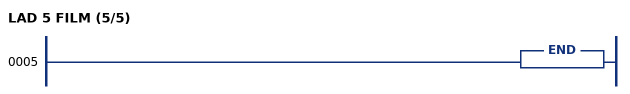
% Rung: 5 %
SOR END EOR

LADDER 6 "PROFILES"
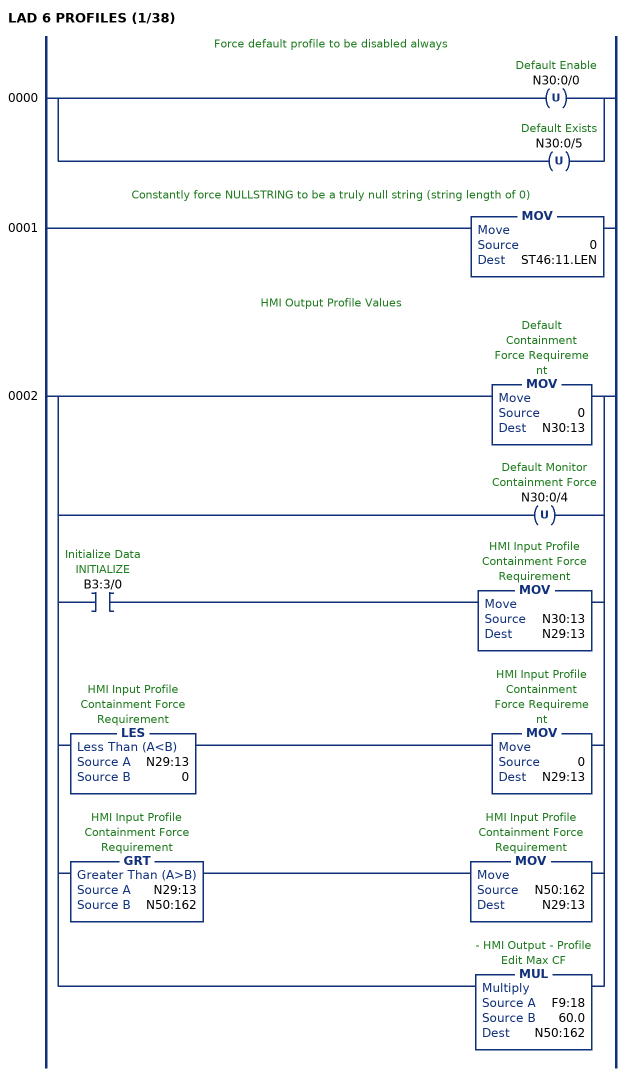
% Rung: 0 %
% Force default profile to be disabled always %
SOR BST OTU N30:0/0 NXB OTU N30:0/5 BND EOR
%   N30:0/0  "Default Enable" %
%   N30:0/5  "Default Exists" %
% Rung: 1 %
% Constantly force NULLSTRING to be a truly null string (string length of 0) %
SOR MOV 0 ST46:11.LEN EOR
% Rung: 2 %
% HMI Output Profile Values %
SOR BST MOV 0 N30:13 NXB OTU N30:0/4 NXB XIC B3:3/0 MOV N30:13 N29:13 NXB LES N29:13 0 MOV 0 N29:13 NXB GRT N29:13 N50:162 MOV N50:162 N29:13 NXB MUL F9:18 60.0 N50:162 BND EOR
%   N30:13  "Default Containment Force Requirement" %
%   N30:0/4  "Default Monitor Containment Force" %
%   B3:3/0  INITIALIZE  "Initialize Data" %
%   N29:13  "HMI Input Profile Containment Force Requirement" %
%   N50:162  "- HMI Output - Profile Edit Max CF" %
%   F9:18  INCREMENTALAT15  "Incremental CF At WF15 For A Given Film Thickness" %

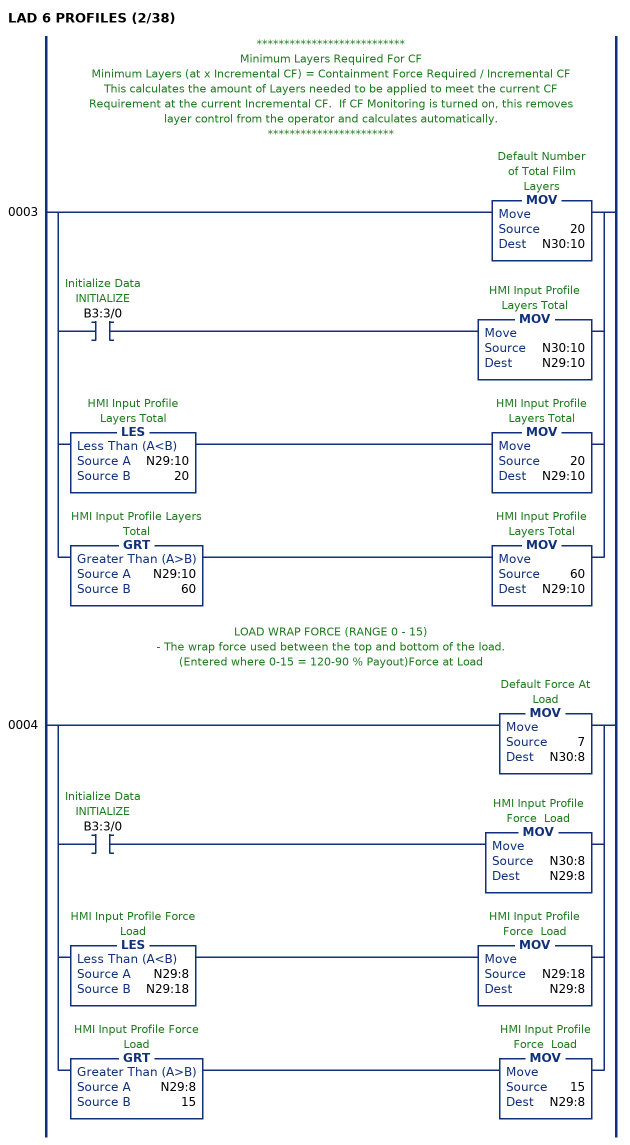
% Rung: 3 %
% ***************************
% 
% Minimum Layers Required For CF
% 
% Minimum Layers (at x Incremental CF) = Containment Force Required / Incremental CF
% 
% This calculates the amount of Layers needed to be applied to meet the current CF Requirement at the current Incremental CF.  If CF Monitoring is turned on, this removes layer control from the operator and calculates automatically.
% 
% *********************** %
SOR BST MOV 20 N30:10 NXB XIC B3:3/0 MOV N30:10 N29:10 NXB LES N29:10 20 MOV 20 N29:10 NXB GRT N29:10 60 MOV 60 N29:10 BND EOR
%   N30:10  "Default Number of Total Film Layers" %
%   B3:3/0  INITIALIZE  "Initialize Data" %
%   N29:10  "HMI Input Profile Layers Total" %
% Rung: 4 %
% LOAD WRAP FORCE (RANGE 0 - 15)
%   - The wrap force used between the top and bottom of the load.
% (Entered where 0-15 = 120-90 % Payout)Force at Load %
SOR BST MOV 7 N30:8 NXB XIC B3:3/0 MOV N30:8 N29:8 NXB LES N29:8 N29:18 MOV N29:18 N29:8 NXB GRT N29:8 15 MOV 15 N29:8 BND EOR
%   N30:8  "Default Force At Load" %
%   B3:3/0  INITIALIZE  "Initialize Data" %
%   N29:8  "HMI Input Profile Force  Load" %
%   N29:18  "HMI Input Profile Force Load Minimum" %

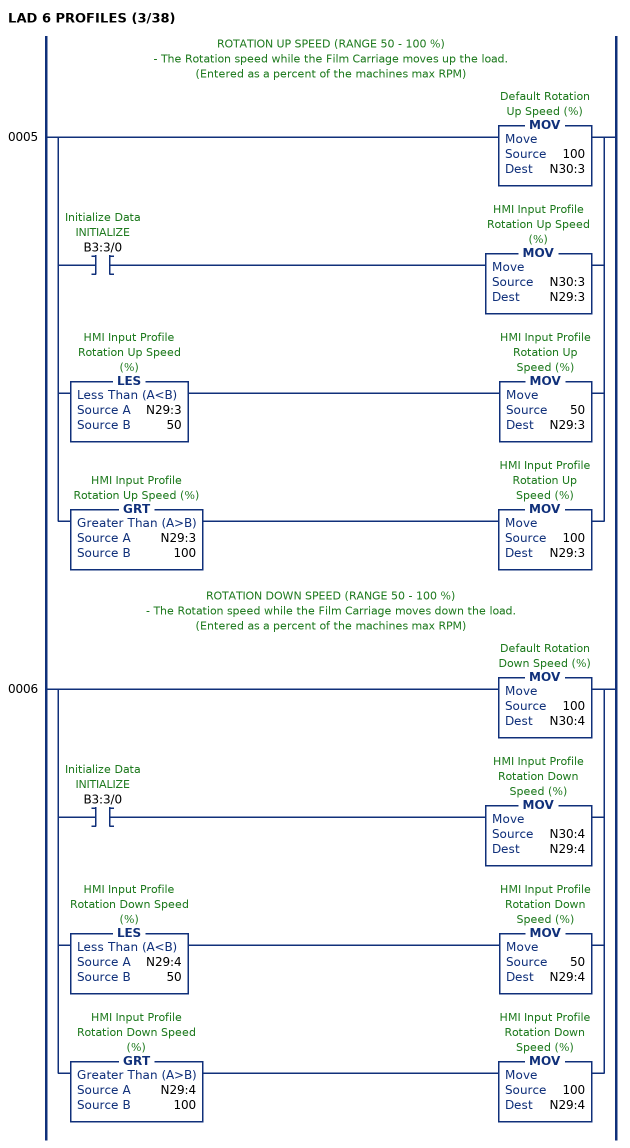
% Rung: 5 %
% ROTATION UP SPEED (RANGE 50 - 100 %)
%   - The Rotation speed while the Film Carriage moves up the load.
% (Entered as a percent of the machines max RPM) %
SOR BST MOV 100 N30:3 NXB XIC B3:3/0 MOV N30:3 N29:3 NXB LES N29:3 50 MOV 50 N29:3 NXB GRT N29:3 100 MOV 100 N29:3 BND EOR
%   N30:3  "Default Rotation Up Speed (%)" %
%   B3:3/0  INITIALIZE  "Initialize Data" %
%   N29:3  "HMI Input Profile Rotation Up Speed (%)" %
% Rung: 6 %
% ROTATION DOWN SPEED (RANGE 50 - 100 %)
%   - The Rotation speed while the Film Carriage moves down the load.
% (Entered as a percent of the machines max RPM) %
SOR BST MOV 100 N30:4 NXB XIC B3:3/0 MOV N30:4 N29:4 NXB LES N29:4 50 MOV 50 N29:4 NXB GRT N29:4 100 MOV 100 N29:4 BND EOR
%   N30:4  "Default Rotation Down Speed (%)" %
%   B3:3/0  INITIALIZE  "Initialize Data" %
%   N29:4  "HMI Input Profile Rotation Down Speed (%)" %

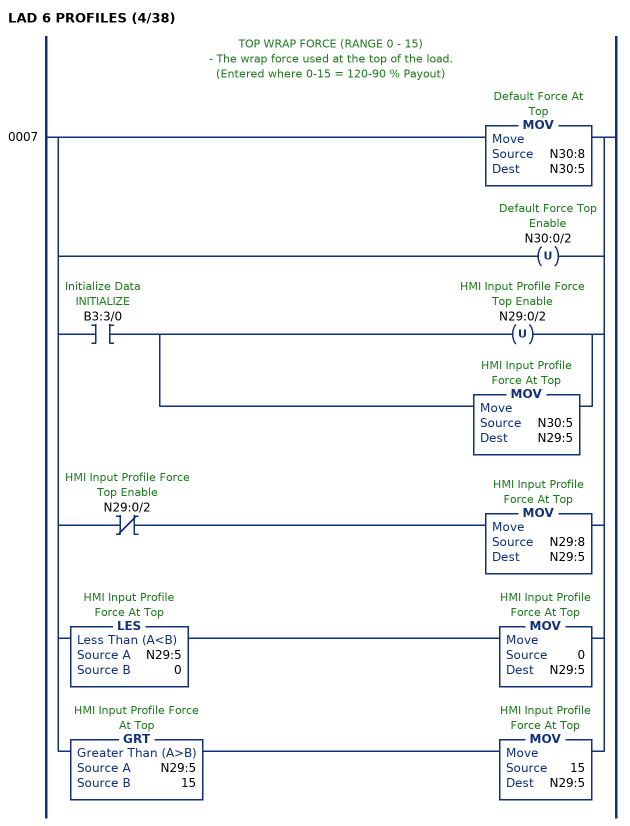
% Rung: 7 %
% TOP WRAP FORCE (RANGE 0 - 15)
%   - The wrap force used at the top of the load.
% (Entered where 0-15 = 120-90 % Payout) %
SOR BST BST MOV N30:8 N30:5 NXB OTU N30:0/2 BND NXB XIC B3:3/0 BST OTU N29:0/2 NXB MOV N30:5 N29:5 BND NXB XIO N29:0/2 MOV N29:8 N29:5 NXB LES N29:5 0 MOV 0 N29:5 NXB GRT N29:5 15 MOV 15 N29:5 BND EOR
%   N30:8  "Default Force At Load" %
%   N30:5  "Default Force At Top" %
%   N30:0/2  "Default Force Top Enable" %
%   B3:3/0  INITIALIZE  "Initialize Data" %
%   N29:0/2  "HMI Input Profile Force Top Enable" %
%   N29:5  "HMI Input Profile Force At Top" %
%   N29:8  "HMI Input Profile Force  Load" %

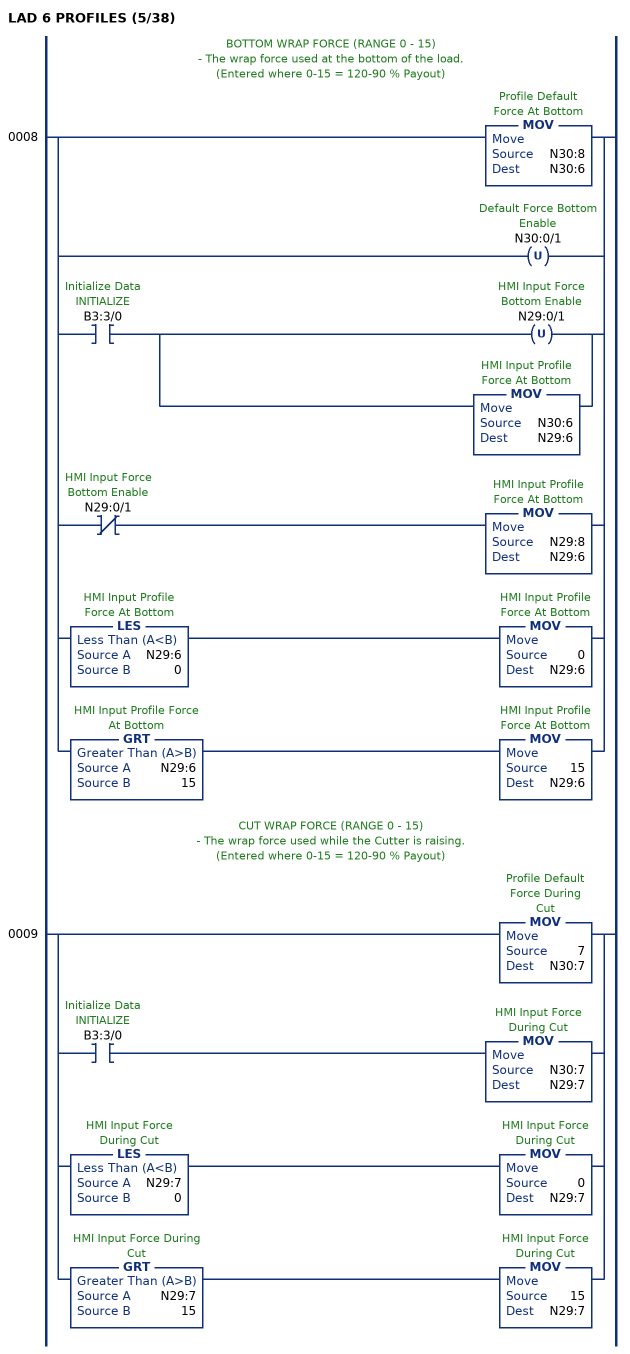
% Rung: 8 %
% BOTTOM WRAP FORCE (RANGE 0 - 15)
%   - The wrap force used at the bottom of the load.
% (Entered where 0-15 = 120-90 % Payout) %
SOR BST BST MOV N30:8 N30:6 NXB OTU N30:0/1 BND NXB XIC B3:3/0 BST OTU N29:0/1 NXB MOV N30:6 N29:6 BND NXB XIO N29:0/1 MOV N29:8 N29:6 NXB LES N29:6 0 MOV 0 N29:6 NXB GRT N29:6 15 MOV 15 N29:6 BND EOR
%   N30:8  "Default Force At Load" %
%   N30:6  "Profile Default Force At Bottom" %
%   N30:0/1  "Default Force Bottom Enable" %
%   B3:3/0  INITIALIZE  "Initialize Data" %
%   N29:0/1  "HMI Input Force Bottom Enable" %
%   N29:6  "HMI Input Profile Force At Bottom" %
%   N29:8  "HMI Input Profile Force  Load" %
% Rung: 9 %
% CUT WRAP FORCE (RANGE 0 - 15)
%   - The wrap force used while the Cutter is raising.
% (Entered where 0-15 = 120-90 % Payout) %
SOR BST MOV 7 N30:7 NXB XIC B3:3/0 MOV N30:7 N29:7 NXB LES N29:7 0 MOV 0 N29:7 NXB GRT N29:7 15 MOV 15 N29:7 BND EOR
%   N30:7  "Profile Default Force During Cut" %
%   B3:3/0  INITIALIZE  "Initialize Data" %
%   N29:7  "HMI Input Force During Cut" %

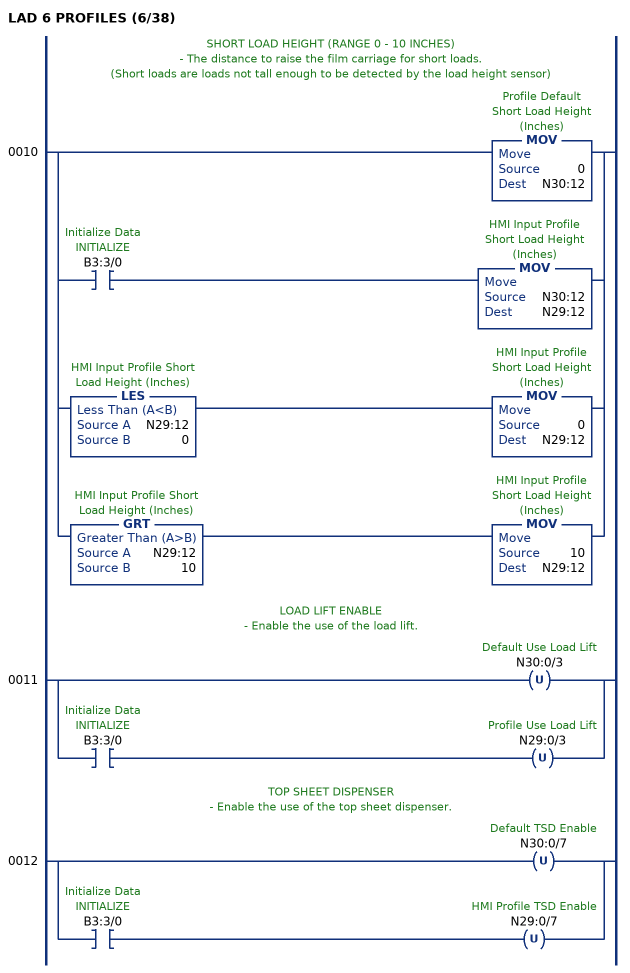
% Rung: 10 %
% SHORT LOAD HEIGHT (RANGE 0 - 10 INCHES)
%   - The distance to raise the film carriage for short loads.
% (Short loads are loads not tall enough to be detected by the load height sensor) %
SOR BST MOV 0 N30:12 NXB XIC B3:3/0 MOV N30:12 N29:12 NXB LES N29:12 0 MOV 0 N29:12 NXB GRT N29:12 10 MOV 10 N29:12 BND EOR
%   N30:12  "Profile Default Short Load Height (Inches)" %
%   B3:3/0  INITIALIZE  "Initialize Data" %
%   N29:12  "HMI Input Profile Short Load Height (Inches)" %
% Rung: 11 %
% LOAD LIFT ENABLE
% - Enable the use of the load lift. %
SOR BST OTU N30:0/3 NXB XIC B3:3/0 OTU N29:0/3 BND EOR
%   N30:0/3  "Default Use Load Lift" %
%   B3:3/0  INITIALIZE  "Initialize Data" %
%   N29:0/3  "Profile Use Load Lift" %
% Rung: 12 %
% TOP SHEET DISPENSER
% - Enable the use of the top sheet dispenser. %
SOR BST OTU N30:0/7 NXB XIC B3:3/0 OTU N29:0/7 BND EOR
%   N30:0/7  "Default TSD Enable" %
%   B3:3/0  INITIALIZE  "Initialize Data" %
%   N29:0/7  "HMI Profile TSD Enable" %

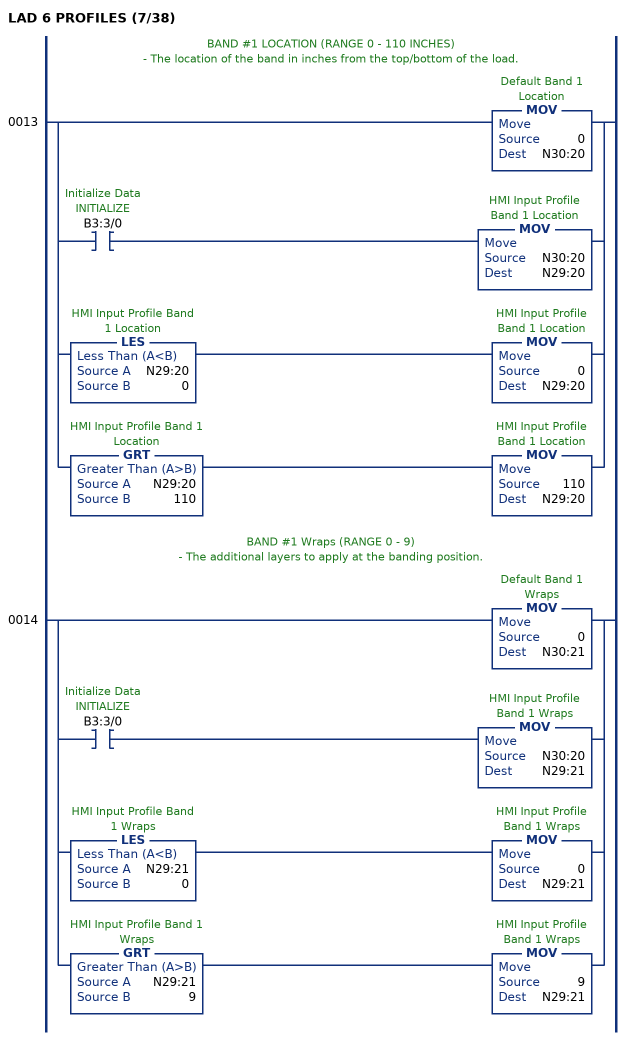
% Rung: 13 %
% BAND #1 LOCATION (RANGE 0 - 110 INCHES)
%   - The location of the band in inches from the top/bottom of the load. %
SOR BST MOV 0 N30:20 NXB XIC B3:3/0 MOV N30:20 N29:20 NXB LES N29:20 0 MOV 0 N29:20 NXB GRT N29:20 110 MOV 110 N29:20 BND EOR
%   N30:20  "Default Band 1 Location" %
%   B3:3/0  INITIALIZE  "Initialize Data" %
%   N29:20  "HMI Input Profile Band 1 Location" %
% Rung: 14 %
% BAND #1 Wraps (RANGE 0 - 9)
%   - The additional layers to apply at the banding position. %
SOR BST MOV 0 N30:21 NXB XIC B3:3/0 MOV N30:20 N29:21 NXB LES N29:21 0 MOV 0 N29:21 NXB GRT N29:21 9 MOV 9 N29:21 BND EOR
%   N30:21  "Default Band 1 Wraps" %
%   B3:3/0  INITIALIZE  "Initialize Data" %
%   N30:20  "Default Band 1 Location" %
%   N29:21  "HMI Input Profile Band 1 Wraps" %

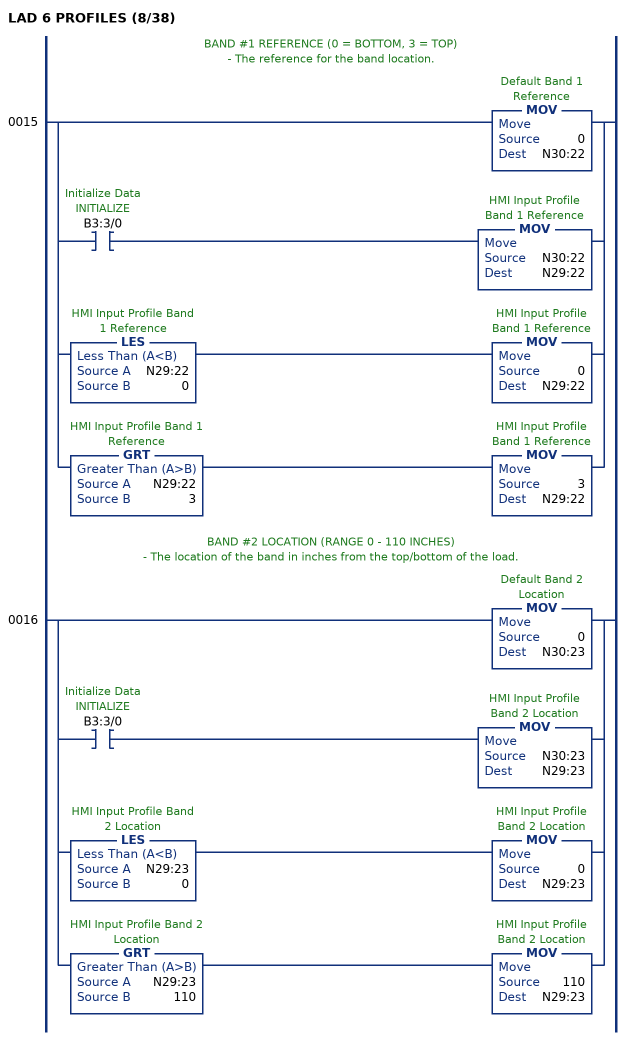
% Rung: 15 %
% BAND #1 REFERENCE (0 = BOTTOM, 3 = TOP)
%   - The reference for the band location. %
SOR BST MOV 0 N30:22 NXB XIC B3:3/0 MOV N30:22 N29:22 NXB LES N29:22 0 MOV 0 N29:22 NXB GRT N29:22 3 MOV 3 N29:22 BND EOR
%   N30:22  "Default Band 1 Reference" %
%   B3:3/0  INITIALIZE  "Initialize Data" %
%   N29:22  "HMI Input Profile Band 1 Reference" %
% Rung: 16 %
% BAND #2 LOCATION (RANGE 0 - 110 INCHES)
%   - The location of the band in inches from the top/bottom of the load. %
SOR BST MOV 0 N30:23 NXB XIC B3:3/0 MOV N30:23 N29:23 NXB LES N29:23 0 MOV 0 N29:23 NXB GRT N29:23 110 MOV 110 N29:23 BND EOR
%   N30:23  "Default Band 2 Location" %
%   B3:3/0  INITIALIZE  "Initialize Data" %
%   N29:23  "HMI Input Profile Band 2 Location" %

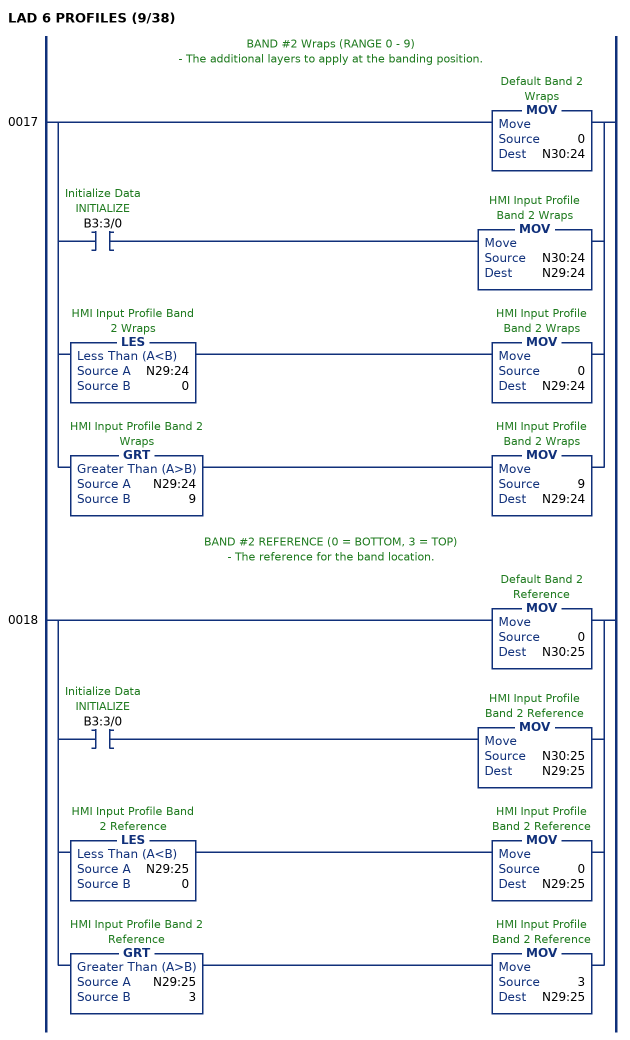
% Rung: 17 %
% BAND #2 Wraps (RANGE 0 - 9)
%   - The additional layers to apply at the banding position. %
SOR BST MOV 0 N30:24 NXB XIC B3:3/0 MOV N30:24 N29:24 NXB LES N29:24 0 MOV 0 N29:24 NXB GRT N29:24 9 MOV 9 N29:24 BND EOR
%   N30:24  "Default Band 2 Wraps" %
%   B3:3/0  INITIALIZE  "Initialize Data" %
%   N29:24  "HMI Input Profile Band 2 Wraps" %
% Rung: 18 %
% BAND #2 REFERENCE (0 = BOTTOM, 3 = TOP)
%   - The reference for the band location. %
SOR BST MOV 0 N30:25 NXB XIC B3:3/0 MOV N30:25 N29:25 NXB LES N29:25 0 MOV 0 N29:25 NXB GRT N29:25 3 MOV 3 N29:25 BND EOR
%   N30:25  "Default Band 2 Reference" %
%   B3:3/0  INITIALIZE  "Initialize Data" %
%   N29:25  "HMI Input Profile Band 2 Reference" %

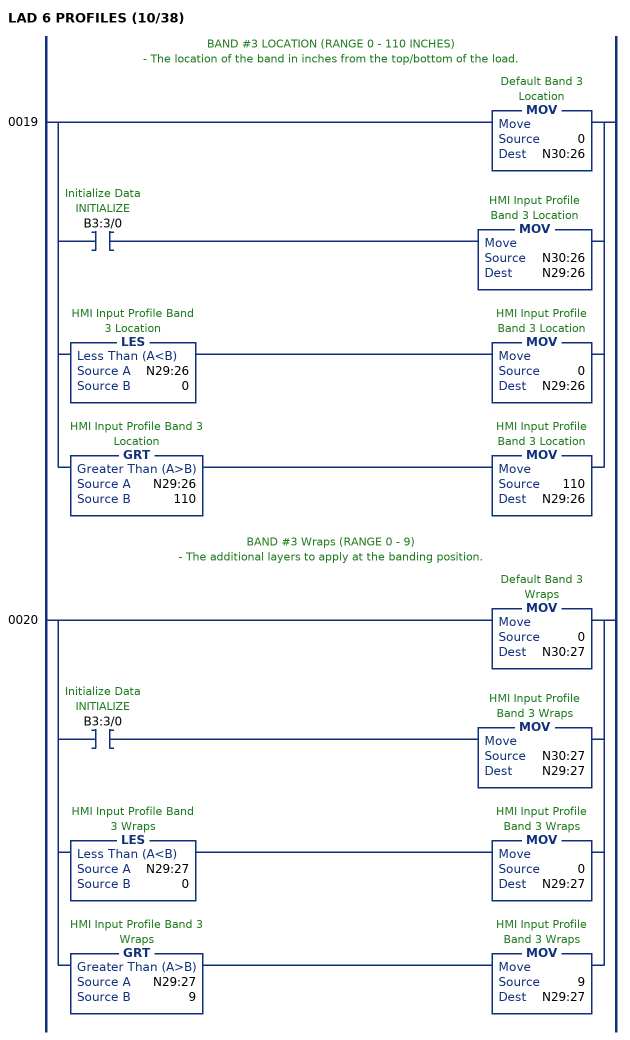
% Rung: 19 %
% BAND #3 LOCATION (RANGE 0 - 110 INCHES)
%   - The location of the band in inches from the top/bottom of the load. %
SOR BST MOV 0 N30:26 NXB XIC B3:3/0 MOV N30:26 N29:26 NXB LES N29:26 0 MOV 0 N29:26 NXB GRT N29:26 110 MOV 110 N29:26 BND EOR
%   N30:26  "Default Band 3 Location" %
%   B3:3/0  INITIALIZE  "Initialize Data" %
%   N29:26  "HMI Input Profile Band 3 Location" %
% Rung: 20 %
% BAND #3 Wraps (RANGE 0 - 9)
%   - The additional layers to apply at the banding position. %
SOR BST MOV 0 N30:27 NXB XIC B3:3/0 MOV N30:27 N29:27 NXB LES N29:27 0 MOV 0 N29:27 NXB GRT N29:27 9 MOV 9 N29:27 BND EOR
%   N30:27  "Default Band 3 Wraps" %
%   B3:3/0  INITIALIZE  "Initialize Data" %
%   N29:27  "HMI Input Profile Band 3 Wraps" %

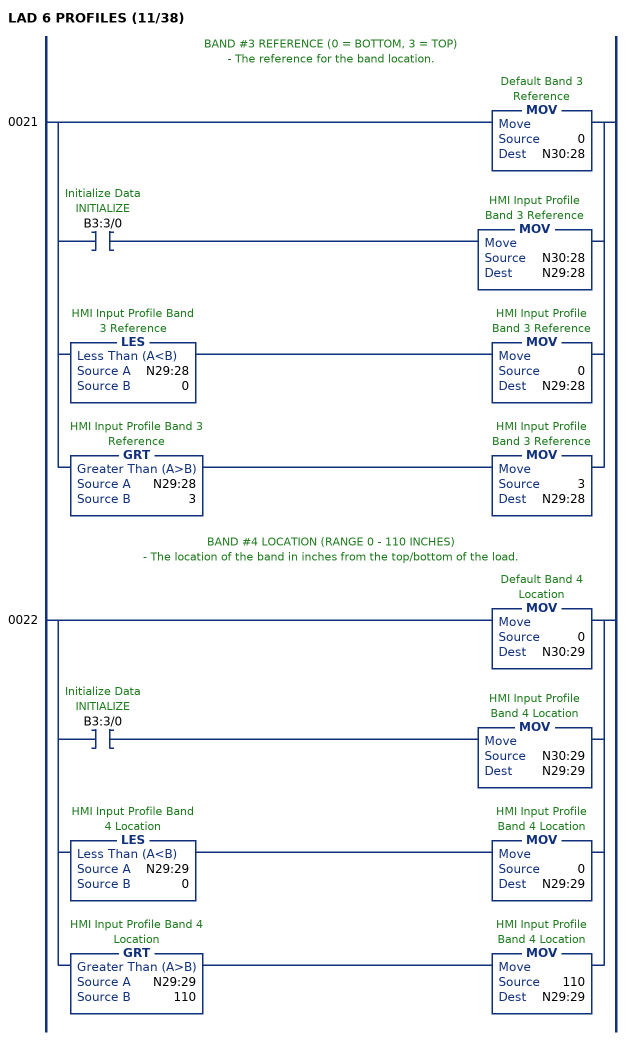
% Rung: 21 %
% BAND #3 REFERENCE (0 = BOTTOM, 3 = TOP)
%   - The reference for the band location. %
SOR BST MOV 0 N30:28 NXB XIC B3:3/0 MOV N30:28 N29:28 NXB LES N29:28 0 MOV 0 N29:28 NXB GRT N29:28 3 MOV 3 N29:28 BND EOR
%   N30:28  "Default Band 3 Reference" %
%   B3:3/0  INITIALIZE  "Initialize Data" %
%   N29:28  "HMI Input Profile Band 3 Reference" %
% Rung: 22 %
% BAND #4 LOCATION (RANGE 0 - 110 INCHES)
%   - The location of the band in inches from the top/bottom of the load. %
SOR BST MOV 0 N30:29 NXB XIC B3:3/0 MOV N30:29 N29:29 NXB LES N29:29 0 MOV 0 N29:29 NXB GRT N29:29 110 MOV 110 N29:29 BND EOR
%   N30:29  "Default Band 4 Location" %
%   B3:3/0  INITIALIZE  "Initialize Data" %
%   N29:29  "HMI Input Profile Band 4 Location" %

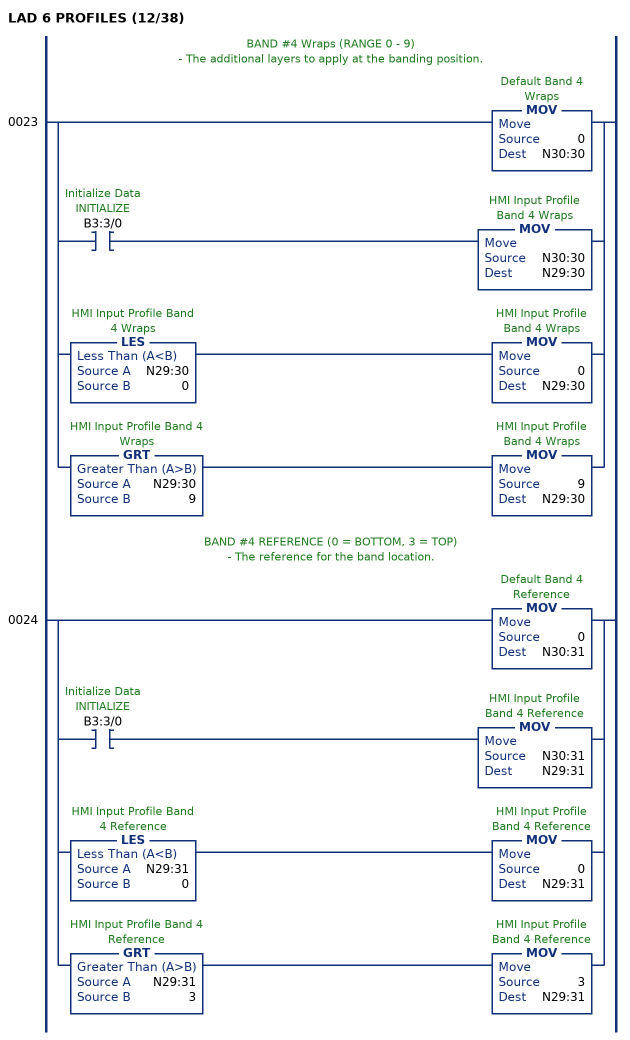
% Rung: 23 %
% BAND #4 Wraps (RANGE 0 - 9)
%   - The additional layers to apply at the banding position. %
SOR BST MOV 0 N30:30 NXB XIC B3:3/0 MOV N30:30 N29:30 NXB LES N29:30 0 MOV 0 N29:30 NXB GRT N29:30 9 MOV 9 N29:30 BND EOR
%   N30:30  "Default Band 4 Wraps" %
%   B3:3/0  INITIALIZE  "Initialize Data" %
%   N29:30  "HMI Input Profile Band 4 Wraps" %
% Rung: 24 %
% BAND #4 REFERENCE (0 = BOTTOM, 3 = TOP)
%   - The reference for the band location. %
SOR BST MOV 0 N30:31 NXB XIC B3:3/0 MOV N30:31 N29:31 NXB LES N29:31 0 MOV 0 N29:31 NXB GRT N29:31 3 MOV 3 N29:31 BND EOR
%   N30:31  "Default Band 4 Reference" %
%   B3:3/0  INITIALIZE  "Initialize Data" %
%   N29:31  "HMI Input Profile Band 4 Reference" %

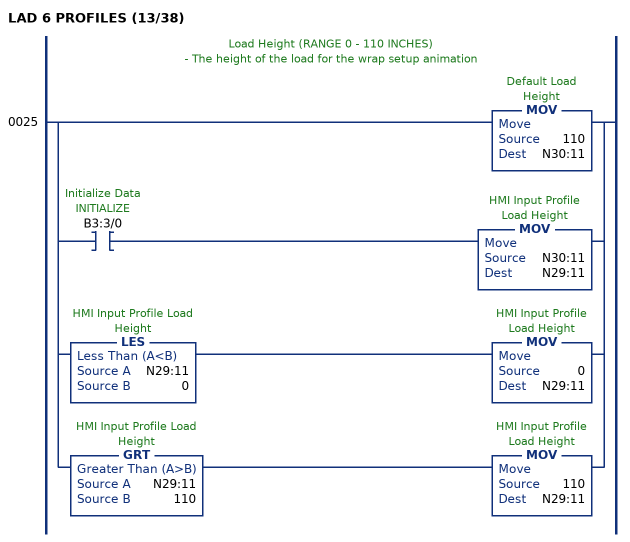
% Rung: 25 %
% Load Height (RANGE 0 - 110 INCHES)
%   - The height of the load for the wrap setup animation %
SOR BST MOV 110 N30:11 NXB XIC B3:3/0 MOV N30:11 N29:11 NXB LES N29:11 0 MOV 0 N29:11 NXB GRT N29:11 110 MOV 110 N29:11 BND EOR
%   N30:11  "Default Load Height" %
%   B3:3/0  INITIALIZE  "Initialize Data" %
%   N29:11  "HMI Input Profile Load Height" %

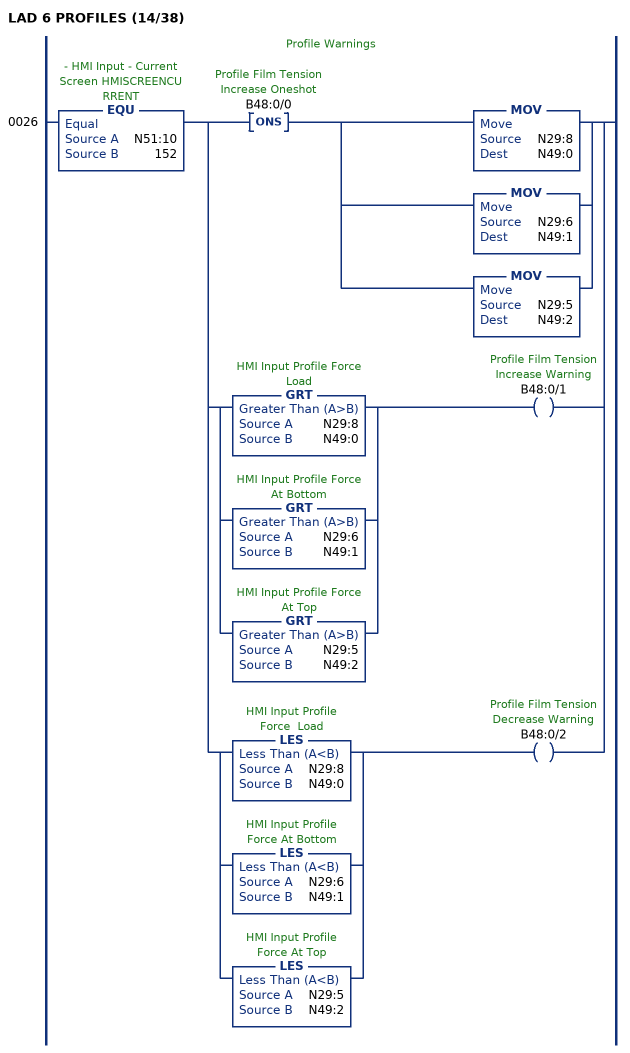
% Rung: 26 %
% Profile Warnings %
SOR EQU N51:10 152 BST ONS B48:0/0 BST MOV N29:8 N49:0 NXB MOV N29:6 N49:1 NXB MOV N29:5 N49:2 BND NXB BST GRT N29:8 N49:0 NXB GRT N29:6 N49:1 NXB GRT N29:5 N49:2 BND OTE B48:0/1 NXB BST LES N29:8 N49:0 NXB LES N29:6 N49:1 NXB LES N29:5 N49:2 BND OTE B48:0/2 BND EOR
%   N51:10  HMISCREENCURRENT  "- HMI Input - Current Screen" %
%   B48:0/0  "Profile Film Tension Increase Oneshot" %
%   N29:8  "HMI Input Profile Force  Load" %
%   N29:6  "HMI Input Profile Force At Bottom" %
%   N29:5  "HMI Input Profile Force At Top" %
%   B48:0/1  "Profile Film Tension Increase Warning" %
%   B48:0/2  "Profile Film Tension Decrease Warning" %

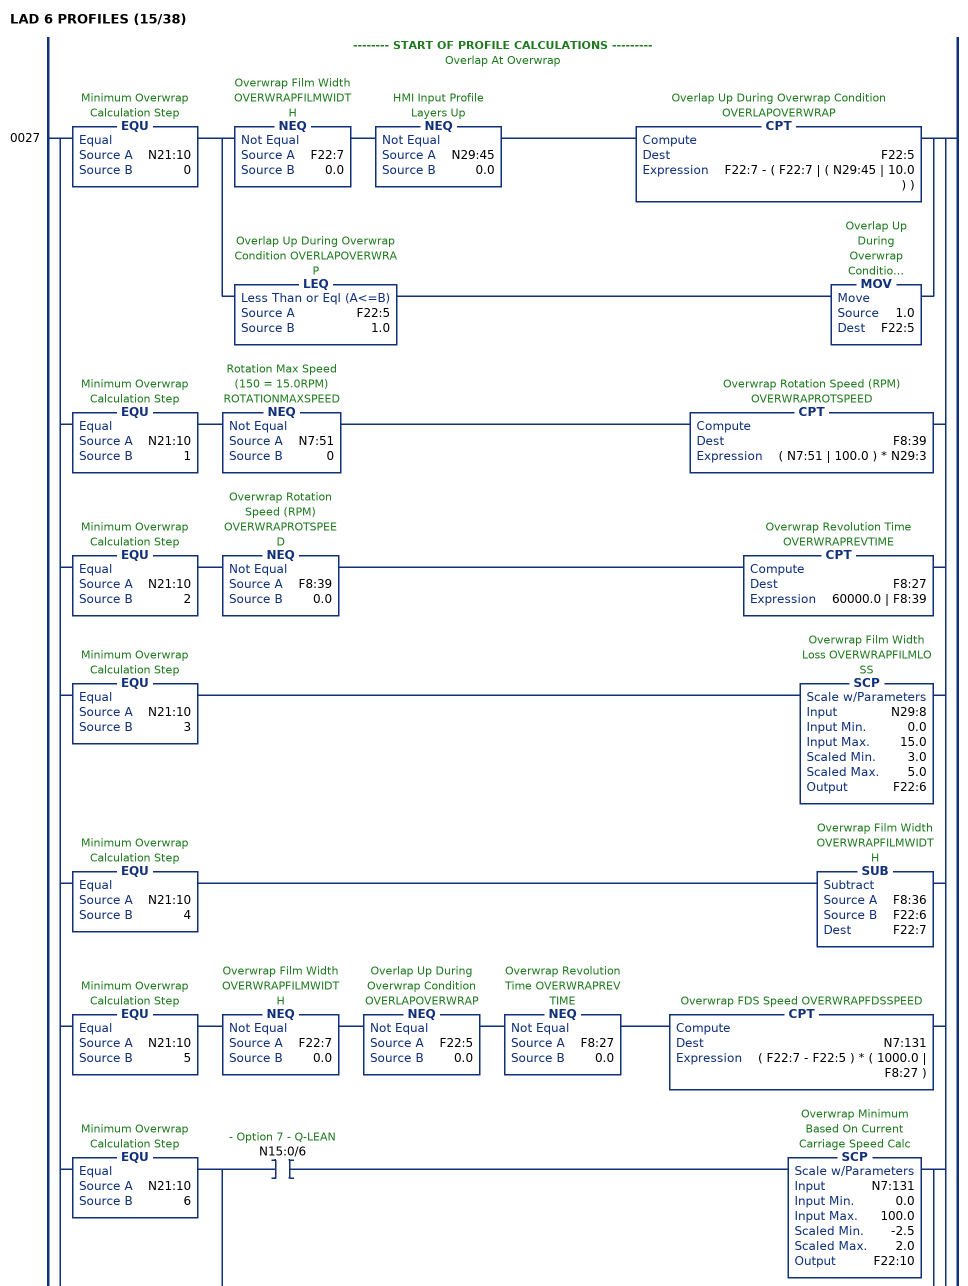

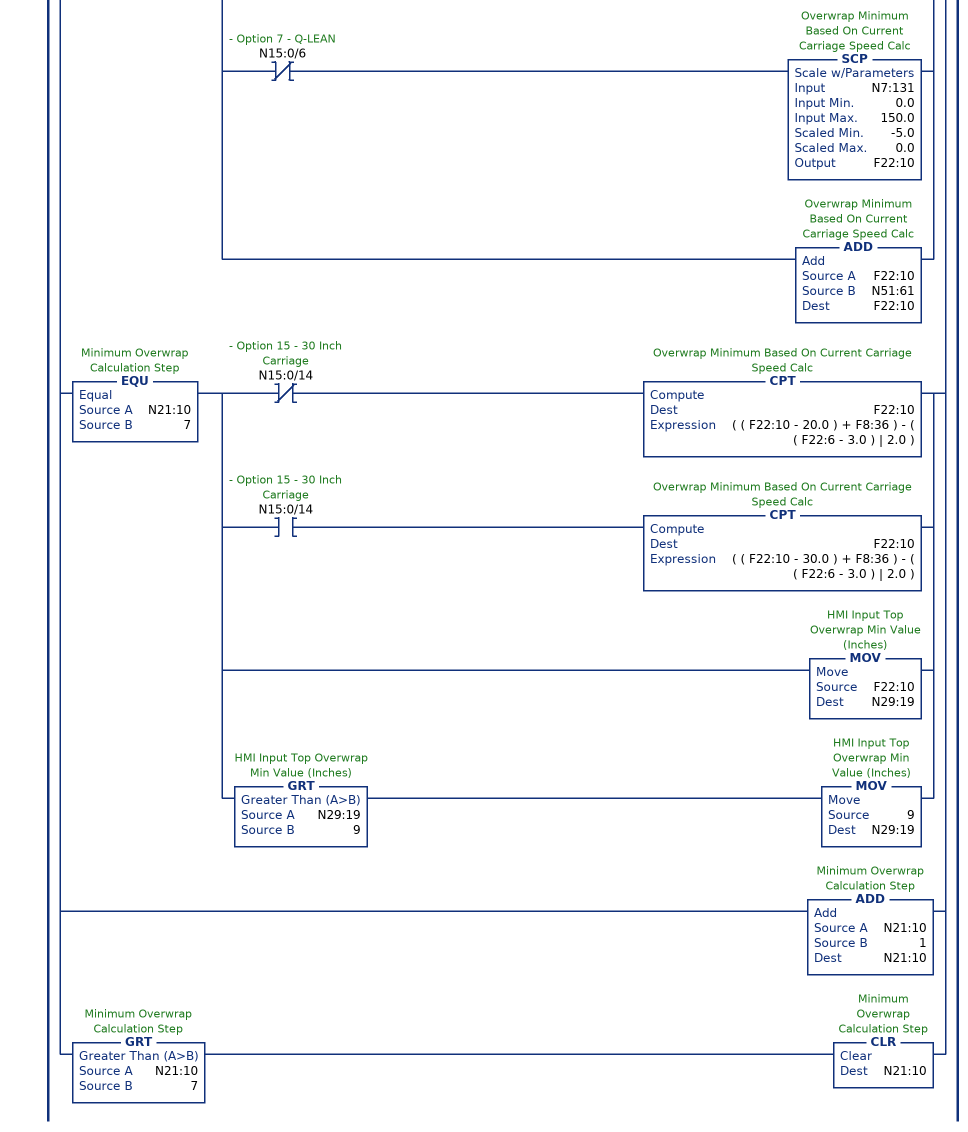
% Rung: 27 %
% TITLE: -------- START OF PROFILE CALCULATIONS --------- %
% Overlap At Overwrap %
SOR BST EQU N21:10 0 BST NEQ F22:7 0.0 NEQ N29:45 0.0 CPT F22:5 " F22:7 - ( F22:7 | ( N29:45 | 10.0 ) ) " NXB LEQ F22:5 1.0 MOV 1.0 F22:5 BND NXB EQU N21:10 1 NEQ N7:51 0 CPT F8:39 " ( N7:51 | 100.0 ) * N29:3 " NXB EQU N21:10 2 NEQ F8:39 0.0 CPT F8:27 " 60000.0 | F8:39 " NXB EQU N21:10 3 SCP N29:8 0.0 15.0 3.0 5.0 F22:6 NXB EQU N21:10 4 SUB F8:36 F22:6 F22:7 NXB EQU N21:10 5 NEQ F22:7 0.0 NEQ F22:5 0.0 NEQ F8:27 0.0 CPT N7:131 " ( F22:7 - F22:5 ) * ( 1000.0 | F8:27 ) " NXB EQU N21:10 6 BST XIC N15:0/6 SCP N7:131 0.0 100.0 -2.5 2.0 F22:10 NXB XIO N15:0/6 SCP N7:131 0.0 150.0 -5.0 0.0 F22:10 NXB ADD F22:10 N51:61 F22:10 BND NXB EQU N21:10 7 BST XIO N15:0/14 CPT F22:10 " ( ( F22:10 - 20.0 ) + F8:36 ) - ( ( F22:6 - 3.0 ) | 2.0 ) " NXB XIC N15:0/14 CPT F22:10 " ( ( F22:10 - 30.0 ) + F8:36 ) - ( ( F22:6 - 3.0 ) | 2.0 ) " NXB BST MOV F22:10 N29:19 NXB GRT N29:19 9 MOV 9 N29:19 BND BND NXB BST ADD N21:10 1 N21:10 NXB GRT N21:10 7 CLR N21:10 BND BND EOR
%   N21:10  "Minimum Overwrap Calculation Step" %
%   F22:7  OVERWRAPFILMWIDTH  "Overwrap Film Width" %
%   N29:45  "HMI Input Profile Layers Up" %
%   F22:5  OVERLAPOVERWRAP  "Overlap Up During Overwrap Condition" %
%   N7:51  ROTATIONMAXSPEED  "Rotation Max Speed (150 = 15.0RPM)" %
%   F8:39  OVERWRAPROTSPEED  "Overwrap Rotation Speed (RPM)" %
%   N29:3  "HMI Input Profile Rotation Up Speed (%)" %
%   F8:27  OVERWRAPREVTIME  "Overwrap Revolution Time" %
%   N29:8  "HMI Input Profile Force  Load" %
%   F22:6  OVERWRAPFILMLOSS  "Overwrap Film Width Loss" %
%   F8:36  FILMSIZE  "Film Size (Inches)" %
%   N7:131  OVERWRAPFDSSPEED  "Overwrap FDS Speed" %
%   N15:0/6  "- Option 7 - Q-LEAN" %
%   F22:10  "Overwrap Minimum Based On Current Carriage Speed Calc" %
%   N51:61  "- HMI Input - Load Height Sensing Offset" %
%   N15:0/14  "- Option 15 - 30 Inch Carriage" %
%   N29:19  "HMI Input Top Overwrap Min Value (Inches)" %

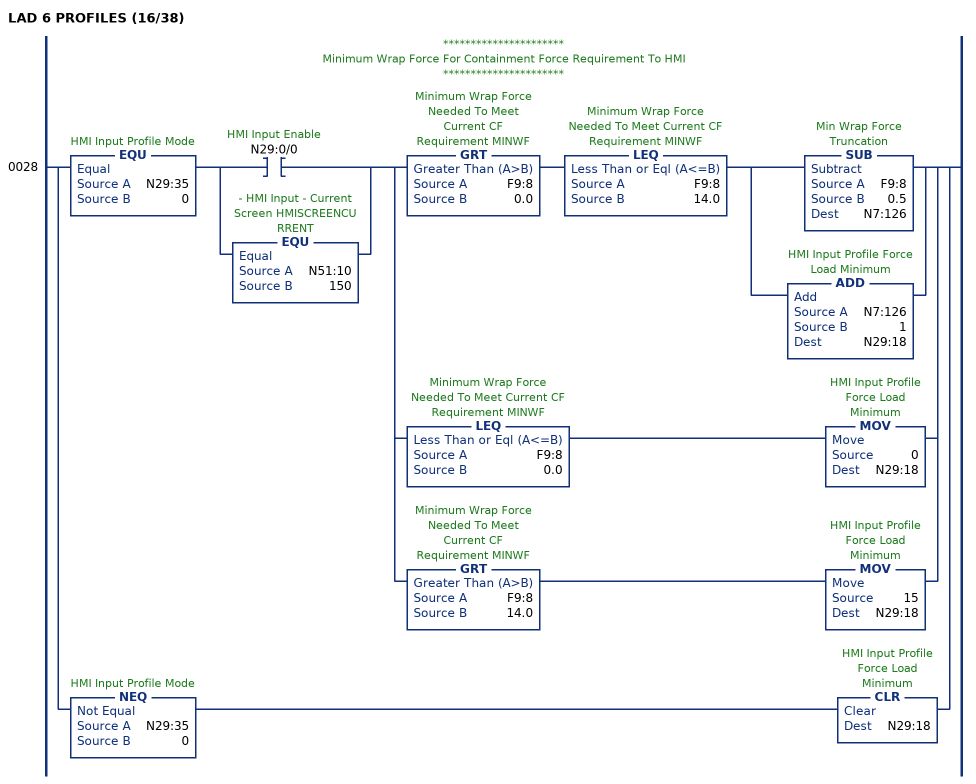
% Rung: 28 %
% **********************
% 
% Minimum Wrap Force For Containment Force Requirement To HMI
% 
% ********************** %
SOR BST EQU N29:35 0 BST XIC N29:0/0 NXB EQU N51:10 150 BND BST GRT F9:8 0.0 LEQ F9:8 14.0 BST SUB F9:8 0.5 N7:126 NXB ADD N7:126 1 N29:18 BND NXB LEQ F9:8 0.0 MOV 0 N29:18 NXB GRT F9:8 14.0 MOV 15 N29:18 BND NXB NEQ N29:35 0 CLR N29:18 BND EOR
%   N29:35  "HMI Input Profile Mode" %
%   N29:0/0  "HMI Input Enable" %
%   N51:10  HMISCREENCURRENT  "- HMI Input - Current Screen" %
%   F9:8  MINWF  "Minimum Wrap Force Needed To Meet Current CF Requirement" %
%   N7:126  "Min Wrap Force Truncation" %
%   N29:18  "HMI Input Profile Force Load Minimum" %

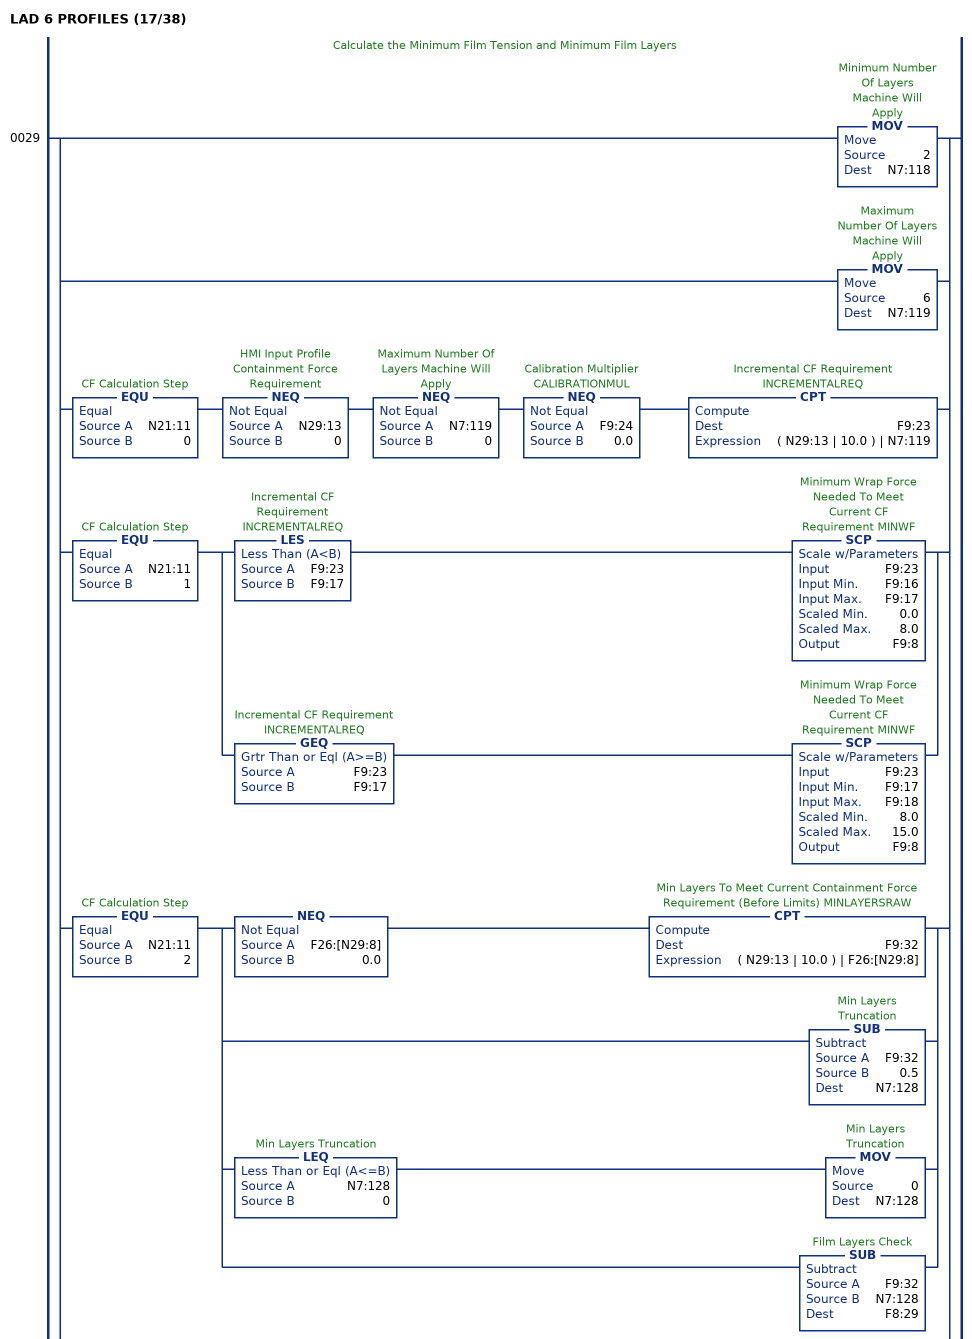

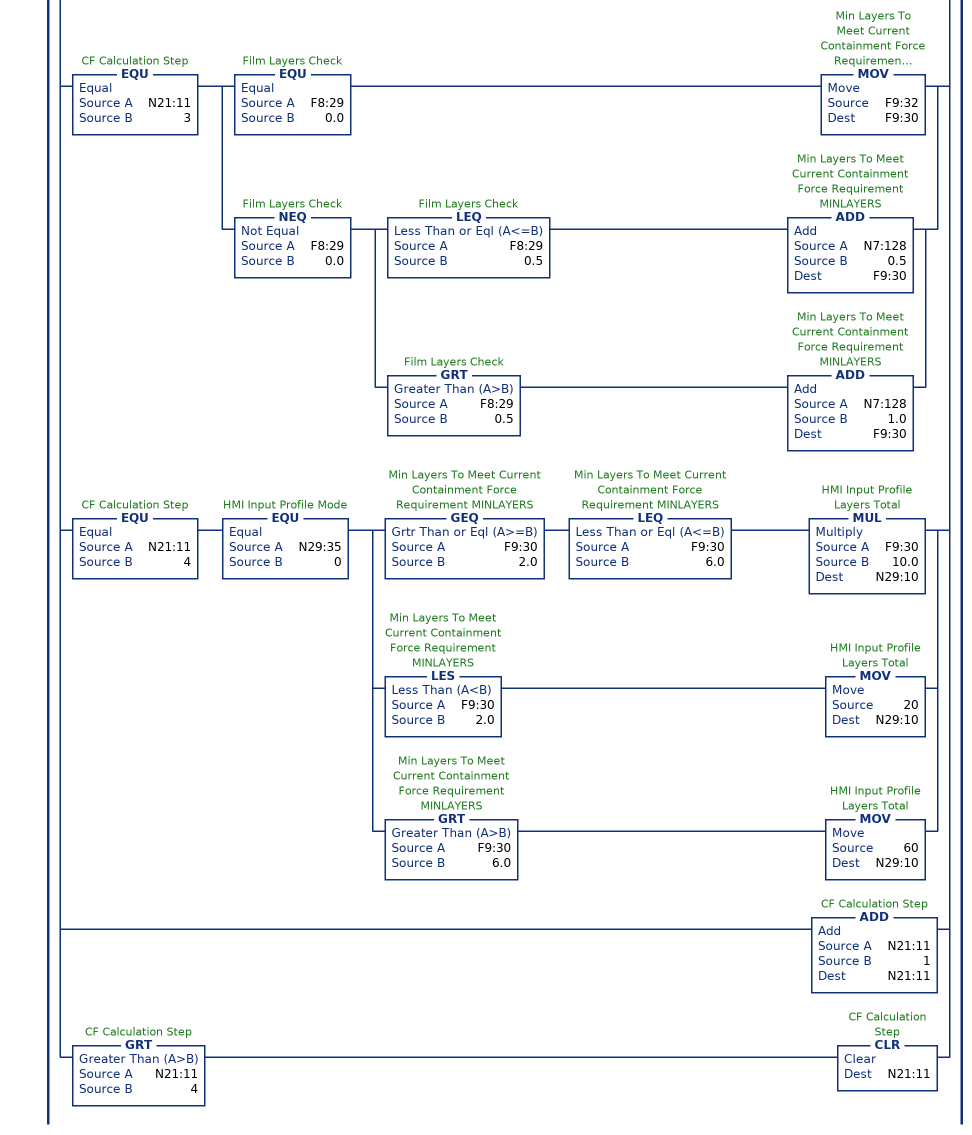
% Rung: 29 %
% Calculate the Minimum Film Tension and Minimum Film Layers %
SOR BST MOV 2 N7:118 NXB MOV 6 N7:119 NXB EQU N21:11 0 NEQ N29:13 0 NEQ N7:119 0 NEQ F9:24 0.0 CPT F9:23 " ( N29:13 | 10.0 ) | N7:119 " NXB EQU N21:11 1 BST LES F9:23 F9:17 SCP F9:23 F9:16 F9:17 0.0 8.0 F9:8 NXB GEQ F9:23 F9:17 SCP F9:23 F9:17 F9:18 8.0 15.0 F9:8 BND NXB EQU N21:11 2 BST NEQ F26:[N29:8] 0.0 CPT F9:32 " ( N29:13 | 10.0 ) | F26:[N29:8] " NXB SUB F9:32 0.5 N7:128 NXB LEQ N7:128 0 MOV 0 N7:128 NXB SUB F9:32 N7:128 F8:29 BND NXB EQU N21:11 3 BST EQU F8:29 0.0 MOV F9:32 F9:30 NXB NEQ F8:29 0.0 BST LEQ F8:29 0.5 ADD N7:128 0.5 F9:30 NXB GRT F8:29 0.5 ADD N7:128 1.0 F9:30 BND BND NXB EQU N21:11 4 EQU N29:35 0 BST GEQ F9:30 2.0 LEQ F9:30 6.0 MUL F9:30 10.0 N29:10 NXB LES F9:30 2.0 MOV 20 N29:10 NXB GRT F9:30 6.0 MOV 60 N29:10 BND NXB BST ADD N21:11 1 N21:11 NXB GRT N21:11 4 CLR N21:11 BND BND EOR
%   N7:118  "Minimum Number Of Layers Machine Will Apply" %
%   N7:119  "Maximum Number Of Layers Machine Will Apply" %
%   N21:11  "CF Calculation Step" %
%   N29:13  "HMI Input Profile Containment Force Requirement" %
%   F9:24  CALIBRATIONMUL  "Calibration Multiplier" %
%   F9:23  INCREMENTALREQ  "Incremental CF Requirement" %
%   F9:17  INCREMENTALAT8  "Incremental CF At WF8 For A Given Film Thickness" %
%   F9:16  INCREMENTALAT0  "Incremental CF At WF0 For A Given Film Thickness" %
%   F9:8  MINWF  "Minimum Wrap Force Needed To Meet Current CF Requirement" %
%   F9:18  INCREMENTALAT15  "Incremental CF At WF15 For A Given Film Thickness" %
%   N29:8  "HMI Input Profile Force  Load" %
%   F9:32  MINLAYERSRAW  "Min Layers To Meet Current Containment Force Requirement (Before Limits)" %
%   N7:128  "Min Layers Truncation" %
%   F8:29  "Film Layers Check" %
%   F9:30  MINLAYERS  "Min Layers To Meet Current Containment Force Requirement" %
%   N29:35  "HMI Input Profile Mode" %
%   N29:10  "HMI Input Profile Layers Total" %

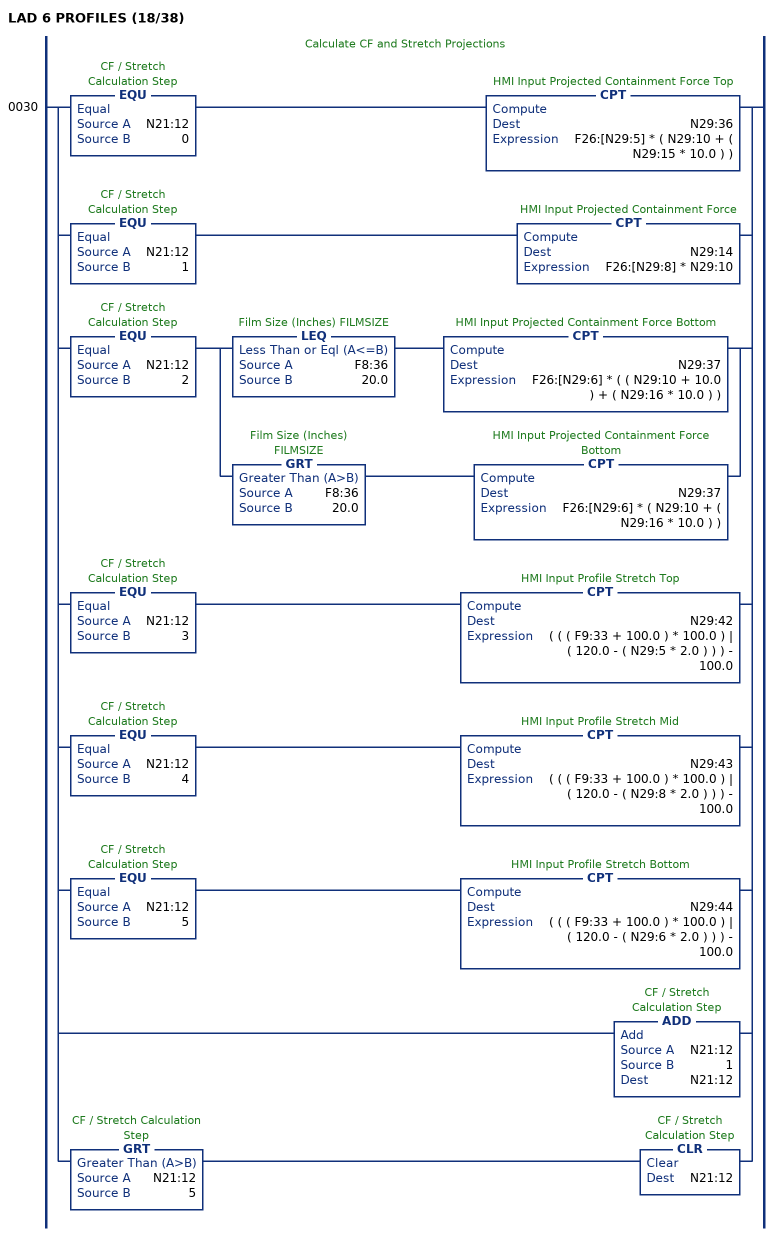
% Rung: 30 %
% Calculate CF and Stretch Projections %
SOR BST EQU N21:12 0 CPT N29:36 " F26:[N29:5] * ( N29:10 + ( N29:15 * 10.0 ) ) " NXB EQU N21:12 1 CPT N29:14 " F26:[N29:8] * N29:10 " NXB EQU N21:12 2 BST LEQ F8:36 20.0 CPT N29:37 " F26:[N29:6] * ( ( N29:10 + 10.0 ) + ( N29:16 * 10.0 ) ) " NXB GRT F8:36 20.0 CPT N29:37 " F26:[N29:6] * ( N29:10 + ( N29:16 * 10.0 ) ) " BND NXB EQU N21:12 3 CPT N29:42 " ( ( ( F9:33 + 100.0 ) * 100.0 ) | ( 120.0 - ( N29:5 * 2.0 ) ) ) - 100.0 " NXB EQU N21:12 4 CPT N29:43 " ( ( ( F9:33 + 100.0 ) * 100.0 ) | ( 120.0 - ( N29:8 * 2.0 ) ) ) - 100.0 " NXB EQU N21:12 5 CPT N29:44 " ( ( ( F9:33 + 100.0 ) * 100.0 ) | ( 120.0 - ( N29:6 * 2.0 ) ) ) - 100.0 " NXB BST ADD N21:12 1 N21:12 NXB GRT N21:12 5 CLR N21:12 BND BND EOR
%   N21:12  "CF / Stretch Calculation Step" %
%   N29:36  "HMI Input Projected Containment Force Top" %
%   N29:5  "HMI Input Profile Force At Top" %
%   N29:10  "HMI Input Profile Layers Total" %
%   N29:14  "HMI Input Projected Containment Force" %
%   N29:8  "HMI Input Profile Force  Load" %
%   F8:36  FILMSIZE  "Film Size (Inches)" %
%   N29:37  "HMI Input Projected Containment Force Bottom" %
%   N29:6  "HMI Input Profile Force At Bottom" %
%   N29:16  "HMI Input Bottom Wraps Adjust" %
%   N29:42  "HMI Input Profile Stretch Top" %
%   F9:33  PRESTRETCH  "Pre-Stretch %" %
%   N29:43  "HMI Input Profile Stretch Mid" %
%   N29:44  "HMI Input Profile Stretch Bottom" %

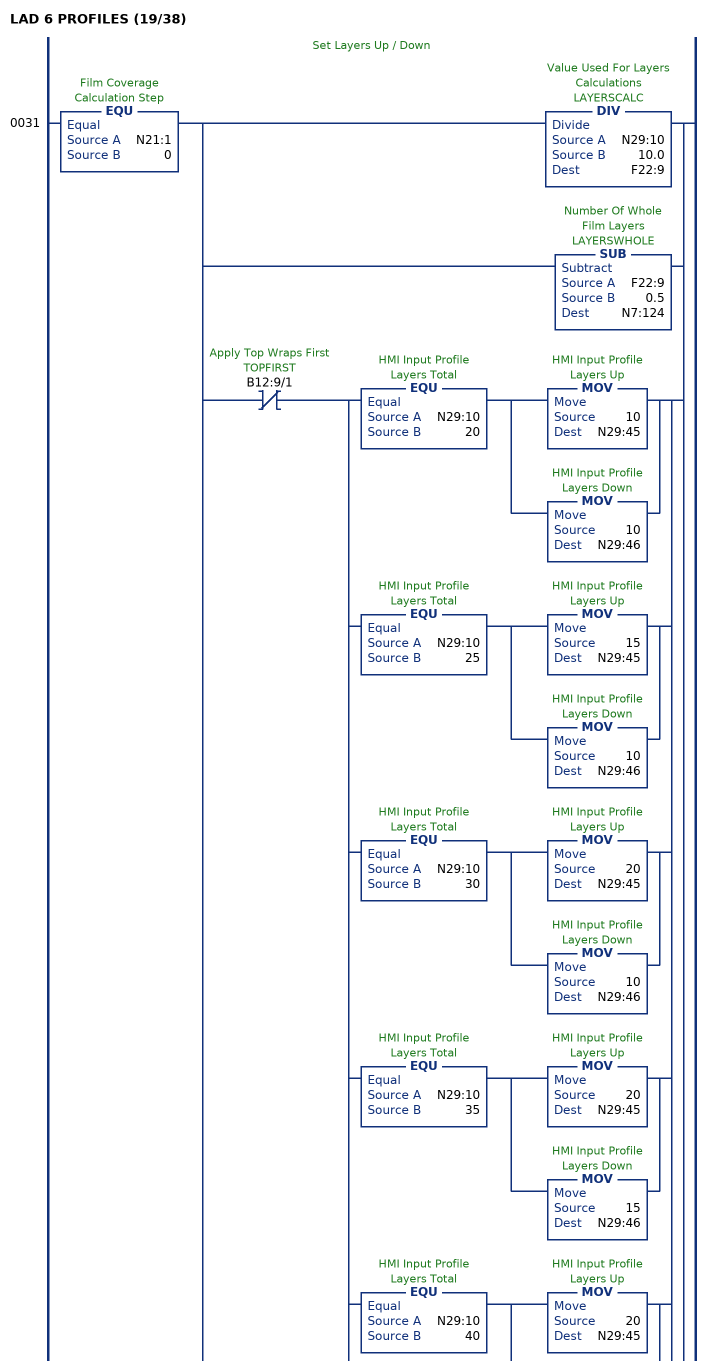

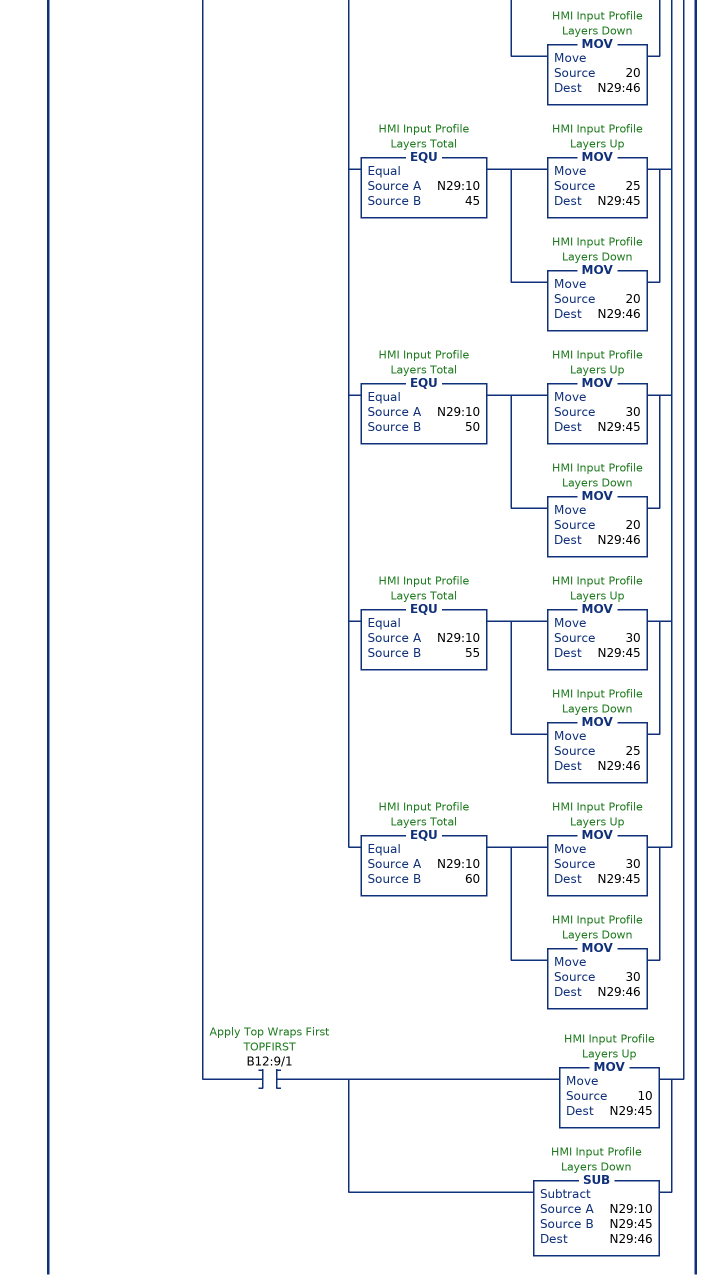
% Rung: 31 %
% Set Layers Up / Down %
SOR EQU N21:1 0 BST DIV N29:10 10.0 F22:9 NXB SUB F22:9 0.5 N7:124 NXB XIO B12:9/1 BST EQU N29:10 20 BST MOV 10 N29:45 NXB MOV 10 N29:46 BND NXB EQU N29:10 25 BST MOV 15 N29:45 NXB MOV 10 N29:46 BND NXB EQU N29:10 30 BST MOV 20 N29:45 NXB MOV 10 N29:46 BND NXB EQU N29:10 35 BST MOV 20 N29:45 NXB MOV 15 N29:46 BND NXB EQU N29:10 40 BST MOV 20 N29:45 NXB MOV 20 N29:46 BND NXB EQU N29:10 45 BST MOV 25 N29:45 NXB MOV 20 N29:46 BND NXB EQU N29:10 50 BST MOV 30 N29:45 NXB MOV 20 N29:46 BND NXB EQU N29:10 55 BST MOV 30 N29:45 NXB MOV 25 N29:46 BND NXB EQU N29:10 60 BST MOV 30 N29:45 NXB MOV 30 N29:46 BND BND NXB XIC B12:9/1 BST MOV 10 N29:45 NXB SUB N29:10 N29:45 N29:46 BND BND EOR
%   N21:1  "Film Coverage Calculation Step" %
%   N29:10  "HMI Input Profile Layers Total" %
%   F22:9  LAYERSCALC  "Value Used For Layers Calculations" %
%   N7:124  LAYERSWHOLE  "Number Of Whole Film Layers" %
%   B12:9/1  TOPFIRST  "Apply Top Wraps First" %
%   N29:45  "HMI Input Profile Layers Up" %
%   N29:46  "HMI Input Profile Layers Down" %

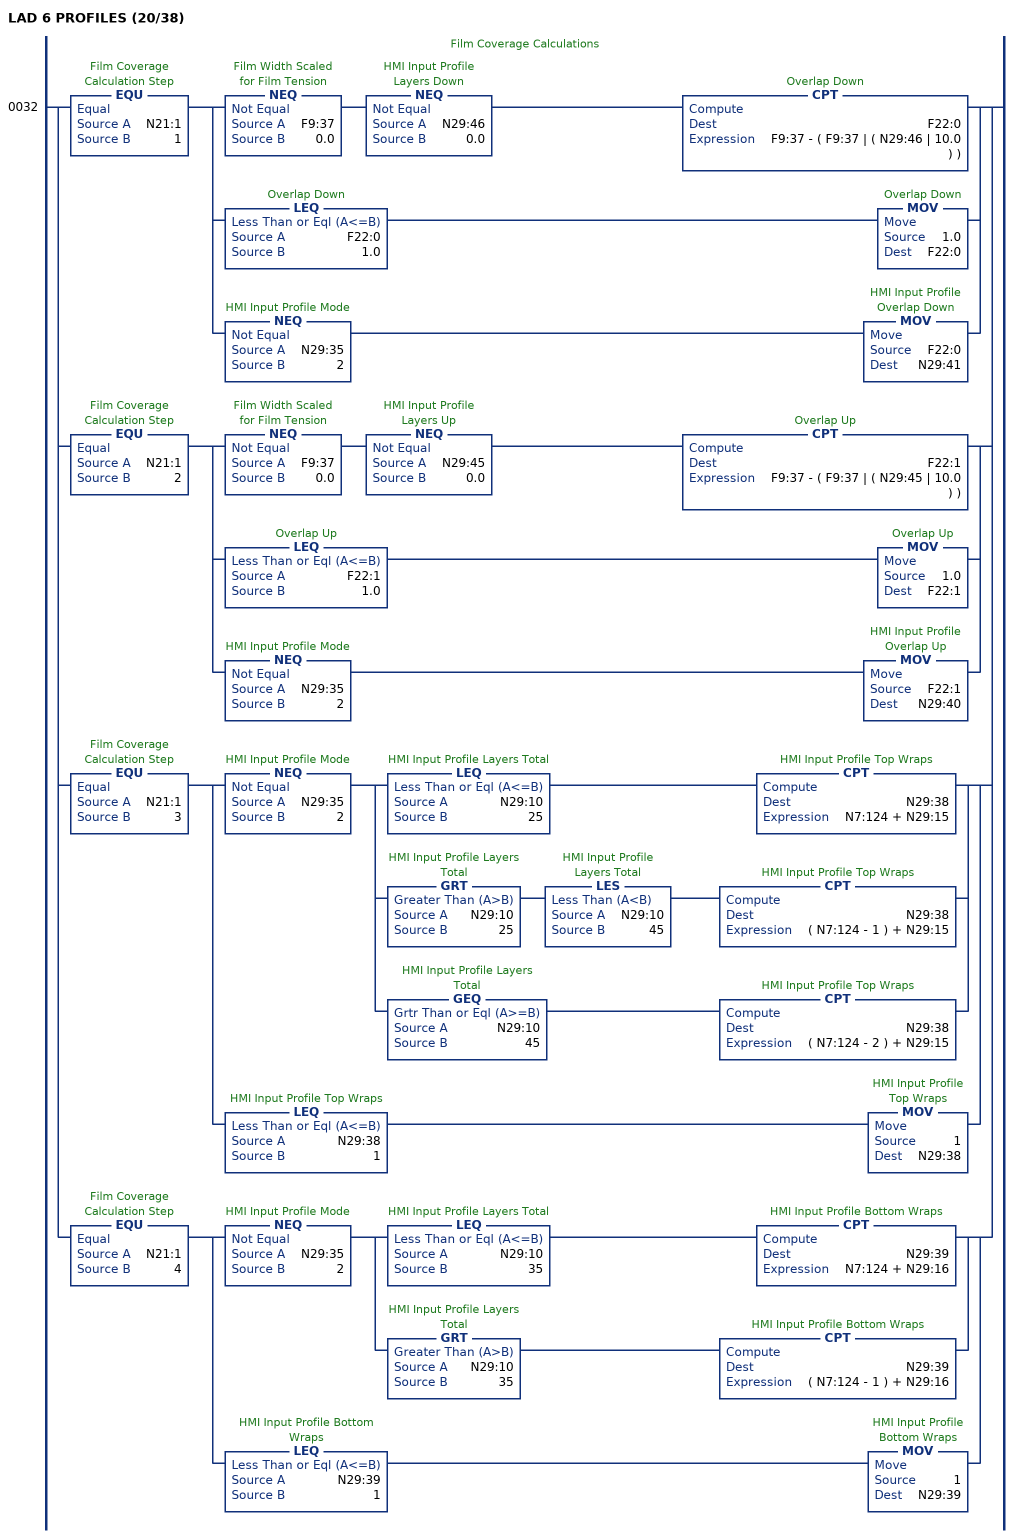
% Rung: 32 %
% Film Coverage Calculations %
SOR BST EQU N21:1 1 BST NEQ F9:37 0.0 NEQ N29:46 0.0 CPT F22:0 " F9:37 - ( F9:37 | ( N29:46 | 10.0 ) ) " NXB LEQ F22:0 1.0 MOV 1.0 F22:0 NXB NEQ N29:35 2 MOV F22:0 N29:41 BND NXB EQU N21:1 2 BST NEQ F9:37 0.0 NEQ N29:45 0.0 CPT F22:1 " F9:37 - ( F9:37 | ( N29:45 | 10.0 ) ) " NXB LEQ F22:1 1.0 MOV 1.0 F22:1 NXB NEQ N29:35 2 MOV F22:1 N29:40 BND NXB EQU N21:1 3 BST NEQ N29:35 2 BST LEQ N29:10 25 CPT N29:38 " N7:124 + N29:15 " NXB GRT N29:10 25 LES N29:10 45 CPT N29:38 " ( N7:124 - 1 ) + N29:15 " NXB GEQ N29:10 45 CPT N29:38 " ( N7:124 - 2 ) + N29:15 " BND NXB LEQ N29:38 1 MOV 1 N29:38 BND NXB EQU N21:1 4 BST NEQ N29:35 2 BST LEQ N29:10 35 CPT N29:39 " N7:124 + N29:16 " NXB GRT N29:10 35 CPT N29:39 " ( N7:124 - 1 ) + N29:16 " BND NXB LEQ N29:39 1 MOV 1 N29:39 BND BND EOR
%   N21:1  "Film Coverage Calculation Step" %
%   F9:37  "Film Width Scaled for Film Tension" %
%   N29:46  "HMI Input Profile Layers Down" %
%   F22:0  "Overlap Down" %
%   N29:35  "HMI Input Profile Mode" %
%   N29:41  "HMI Input Profile Overlap Down" %
%   N29:45  "HMI Input Profile Layers Up" %
%   F22:1  "Overlap Up" %
%   N29:40  "HMI Input Profile Overlap Up" %
%   N29:10  "HMI Input Profile Layers Total" %
%   N29:38  "HMI Input Profile Top Wraps" %
%   N7:124  LAYERSWHOLE  "Number Of Whole Film Layers" %
%   N29:39  "HMI Input Profile Bottom Wraps" %
%   N29:16  "HMI Input Bottom Wraps Adjust" %

